// TwinCAT 3 PLC project Logger
// ProgramVersion: 3.1.4023.0
// libraries:
//   Tc2_Standard, * (Beckhoff Automation GmbH)
//   Tc2_System, * (Beckhoff Automation GmbH)
//   Tc2_Utilities, * (Beckhoff Automation GmbH)
//   Tc3_Module, * (Beckhoff Automation GmbH)
// project tree:
//   / PlcTask.TcTTO
//   POUs/ Logger.TcPOU, MAIN.TcPOU, Notifier.TcPOU, NotifierEvent.TcPOU
// real-time tasks:
//   TASK PlcTask: cycle T#10ms, priority 20, ADS port 350

CONFIGURATION Logger
    RESOURCE PLC ON TwinCAT3
        TASK PlcTask(INTERVAL := T#10ms, PRIORITY := 20);
        PROGRAM MAIN WITH PlcTask : MAIN;
    END_RESOURCE
END_CONFIGURATION

// ---- POUs/MAIN.TcPOU
PROGRAM MAIN
VAR
	
	diStep : DINT;
	bStart : BOOL;
	bStop : BOOL;
	fbRepeatTimer : TON;
	udiCounter : UDINT;
	
	fbLogger : Logger:= (sPathName:='C:\Users\fboid\Documents\ScopeTest\Log.txt');
	fbNotifier : Notifier := (sPathName:='C:\Users\fboid\Documents\ScopeTest\Log.csv');
	fbNotifierEvent : NotifierEvent;
	i : INT;
	bExecute : BOOL;
	uiCounter : UINT:= 0;
	bMotorError : BOOL;
	
END_VAR


//fbRepeatTimer(IN:= , PT:= T#5S, Q=> , ET=> );

fbNotifier(bExecute := bExecute);
fbNotifierEvent(
	CLK:= bMotorError,  
	fbNotifier:= fbNotifier, 
	sModuleName := 'PreHeat',
	sDeviceName := 'Load conveyor',
	sStatus := 'Error',
	sMessage := 'Motor overloaded');

END_PROGRAM

// ---- POUs/Logger.TcPOU
FUNCTION_BLOCK Logger
VAR_INPUT
	bExecute : BOOL;
	sPathName : STRING;
END_VAR
VAR_OUTPUT
END_VAR
VAR
	aBuffer : ARRAY[1..cMaxBufferRange] OF T_MaxString;
	aWorkBuffer : ARRAY[1..cMaxBufferRange] OF T_MaxString;
	aEmptyBuffer : ARRAY[1..cMaxBufferRange] OF T_MaxString; 
	
	fbFileWrite : FB_FileWrite;
	udiBufferCounter : UDINT;
	udiWorkCounter : UDINT;
	hFile : UINT;	
	
	fbFileOpen : FB_FileOpen;
	fbFilePuts : FB_FilePuts;
	fbFileClose : FB_FileClose;
	
	fbGetSystemTime : GETSYSTEMTIME;
	fbRepeatTimer : TON;
	diStep  : DINT;
	i : UDINT;
	bFilePutsIdle : BOOL;
	bExecuteFilePuts : BOOL;
	bInit : BOOL;
END_VAR
VAR CONSTANT
	cMaxBufferRange : UDINT := 1000;
END_VAR

fbFileOpen(
	sNetId:= , 
	sPathName:= sPathName,
	nMode:= FOPEN_MODEAPPEND OR FOPEN_MODETEXT, 
	ePath:= , 
	bExecute:=, 
	tTimeout:= , 
	bBusy=> , 
	bError=> , 
	nErrId=> , 
	hFile=> hFile);

fbFileWrite(
	sNetId:= , 
	hFile:= hFile, 
	pWriteBuff:= ADR(aWorkBuffer) , 
	cbWriteLen:= , 
	bExecute:= , 
	tTimeout:= , 
	bBusy=> , 
	bError=> , 
	nErrId=> , 
	cbWrite=> );

fbFileClose(
	sNetId:= , 
	hFile:= hFile, 
	bExecute:= , 
	tTimeout:= , 
	bBusy=> , 
	bError=> , 
	nErrId=> );
	
fbRepeatTimer(IN:= , PT:= T#2S, Q=> , ET=> );
//fbTime();

IF NOT bInit
THEN
	bInit := TRUE;
	FOR i := 1 TO cMaxBufferRange DO
		aEmptyBuffer[i] := '';
		aBuffer[i] := '';
		aWorkBuffer[i] := '';
	END_FOR
END_IF

IF 			bExecute
	AND  	diStep = 0
THEN
	diStep := 10;
END_IF	

CASE diStep OF
	
	10:
	
		fbFileOpen.bExecute := TRUE;
		fbRepeatTimer.IN := TRUE;
		diStep := 20;
		
	20:
	
		IF 		NOT fbFileOpen.bBusy
			AND NOT fbFIleOpen.bError
		THEN
			fbFileOpen.bExecute := FALSE;
			diStep := 30;
		END_IF
		
	30:
		
		IF udiBufferCounter > 0
		THEN
			udiWorkCounter := udiBufferCounter;
			udiBufferCounter := 0;
			
			aWorkBuffer := aBuffer;
			aBuffer := aEmptyBuffer;
			
			fbFileWrite.cbWriteLen := udiWorkCounter * (SIZEOF(T_MaxString));
			fbFileWrite.bExecute := TRUE;
			
			diStep := 40;
		ELSIF NOT bExecute
		THEN
			diStep := 50;
		END_IF
		
		
	40:
		
		IF NOT fbFileWrite.bBusy
		THEN
			
			fbFileWrite.bExecute := FALSE;
			IF fbRepeatTimer.Q
			THEN
				fbRepeatTImer.IN := FALSE;
				diStep := 50;
			ELSE
				diStep := 30;
			END_IF
			
		END_IF
		
	50:
	
		fbFileClose.bExecute := TRUE;
		diStep := 60;
		
	60: 
	
		IF 		NOT fbFileClose.bBusy
			AND NOT fbFileClose.bError
		THEN
			fbFileClose.bExecute := FALSE;
			IF bExecute 
			THEN
				
				diStep := 10;
			ELSE
				diStep := 0;
			END_IF
			
		END_IF
	
END_CASE

METHOD Write 
VAR_INPUT
	sMessage : T_MaxString;
END_VAR
VAR
	iLen : INT;
	iFillNumber : INT;
	i : INT;
	sTime : STRING;
	fileTime        : T_FILETIME;
END_VAR
IF udiBufferCounter < cMaxBufferRange
THEN

	udiBufferCounter := udiBufferCounter + 1;
	
	fbGetSystemTime(timeLoDW=>fileTime.dwLowDateTime, timeHiDW=>fileTime.dwHighDateTime );
	sTime :=SYSTEMTIME_TO_STRING( FILETIME_TO_SYSTEMTIME( fileTime ) );
	
	aBuffer[udiBufferCounter] := sTime;
	aBuffer[udiBufferCounter] := CONCAT(aBuffer[udiBufferCounter],': ');
	aBuffer[udiBufferCounter] := CONCAT(aBuffer[udiBufferCounter],sMessage);
	
	iLen := LEN(aBuffer[udiBufferCounter]);
	iFillNumber := 254-iLen;
	
	FOR i := 1 TO iFillNumber DO
		aBuffer[udiBufferCounter] := CONCAT(aBuffer[udiBufferCounter],' ');
	END_FOR
	
	aBuffer[udiBufferCounter][255] := F_ToAsc('$N');
	
END_IF
END_METHOD

END_FUNCTION_BLOCK

// ---- POUs/Notifier.TcPOU
FUNCTION_BLOCK Notifier
VAR_INPUT
	bExecute : BOOL;
	sPathName : STRING;
END_VAR
VAR_OUTPUT
END_VAR
VAR
	aBuffer : ARRAY[1..cMaxBufferRange] OF BYTE;
	aWorkBuffer : ARRAY[1..cMaxBufferRange] OF BYTE;
	aEmptyBuffer : ARRAY[1..cMaxBufferRange] OF BYTE; 
	
	fbFileWrite : FB_FileWrite;
	udiBufferCounter : UDINT;
	udiWorkCounter : UDINT;
	hFile : UINT;	
	
	fbFileOpen : FB_FileOpen;
	fbFilePuts : FB_FilePuts;
	fbFileClose : FB_FileClose;
	
	fbGetSystemTime : GETSYSTEMTIME;
	fbRepeatTimer : TON;
	diStep  : DINT;
	i : UDINT;
	bFilePutsIdle : BOOL;
	bExecuteFilePuts : BOOL;
	bInit : BOOL;
END_VAR
VAR CONSTANT
	cMaxBufferRange : UDINT := 1000 * 256;
END_VAR

fbFileOpen(
	sNetId:= , 
	sPathName:= sPathName,
	nMode:= FOPEN_MODEAPPEND OR FOPEN_MODETEXT, 
	ePath:= , 
	bExecute:=, 
	tTimeout:= , 
	bBusy=> , 
	bError=> , 
	nErrId=> , 
	hFile=> hFile);

fbFileWrite(
	sNetId:= , 
	hFile:= hFile, 
	pWriteBuff:= ADR(aWorkBuffer) , 
	cbWriteLen:= , 
	bExecute:= , 
	tTimeout:= , 
	bBusy=> , 
	bError=> , 
	nErrId=> , 
	cbWrite=> );

fbFileClose(
	sNetId:= , 
	hFile:= hFile, 
	bExecute:= , 
	tTimeout:= , 
	bBusy=> , 
	bError=> , 
	nErrId=> );
	
fbRepeatTimer(IN:= , PT:= T#2S, Q=> , ET=> );
//fbTime();

IF NOT bInit
THEN
	bInit := TRUE;
	(*
	FOR i := 1 TO cMaxBufferRange DO
		aEmptyBuffer[i] := '';
		aBuffer[i] := '';
		aWorkBuffer[i] := '';
	END_FOR
	*)
END_IF

IF 			bExecute
	AND  	diStep = 0
THEN
	diStep := 10;
END_IF	

CASE diStep OF
	
	10:
	
		fbFileOpen.bExecute := TRUE;
		fbRepeatTimer.IN := TRUE;
		diStep := 20;
		
	20:
	
		IF 		NOT fbFileOpen.bBusy
			AND NOT fbFIleOpen.bError
		THEN
			fbFileOpen.bExecute := FALSE;
			diStep := 30;
		END_IF
		
	30:
		
		IF udiBufferCounter > 0
		THEN
			udiWorkCounter := udiBufferCounter-1;
			udiBufferCounter := 0;
			
			aWorkBuffer := aBuffer;
			aBuffer := aEmptyBuffer;
			
			fbFileWrite.cbWriteLen := udiWorkCounter;
			fbFileWrite.bExecute := TRUE;
			
			diStep := 40;
		ELSIF NOT bExecute
		THEN
			diStep := 50;
		END_IF
		
		
	40:
		
		IF NOT fbFileWrite.bBusy
		THEN
			
			fbFileWrite.bExecute := FALSE;
			IF fbRepeatTimer.Q
			THEN
				fbRepeatTImer.IN := FALSE;
				diStep := 50;
			ELSE
				diStep := 30;
			END_IF
			
		END_IF
		
	50:
	
		fbFileClose.bExecute := TRUE;
		diStep := 60;
		
	60: 
	
		IF 		NOT fbFileClose.bBusy
			AND NOT fbFileClose.bError
		THEN
			fbFileClose.bExecute := FALSE;
			IF bExecute 
			THEN
				
				diStep := 10;
			ELSE
				diStep := 0;
			END_IF
			
		END_IF
	
END_CASE

METHOD Write 
VAR_INPUT
	
	sModuleName : T_MaxString;
	sDeviceName : T_MaxString;
	sStatus	: T_MaxString;
	sMessage : T_MaxString;
	
END_VAR
VAR
	iLen : INT;
	iFillNumber : INT;
	i : INT;
	sTime : STRING;
	fileTime : T_FILETIME;
	iTmpSize : INT;
	aLocalBuffer : ARRAY[0..MAX_STRING_LENGTH] OF BYTE;
	aEmptyLocalBuffer : ARRAY[0..MAX_STRING_LENGTH] OF BYTE;
END_VAR
IF udiBufferCounter < cMaxBufferRange
THEN
		
	fbGetSystemTime(timeLoDW=>fileTime.dwLowDateTime, timeHiDW=>fileTime.dwHighDateTime );
	sTime :=SYSTEMTIME_TO_STRING( FILETIME_TO_SYSTEMTIME( fileTime ) );

//Insert TimeStamp	
//----------------------------------------------------------------------------------------------------------------------------	
	iTmpSize := LEN(sTime);
	aLocalBuffer := MAXSTRING_TO_BYTEARR(sTime);
	
	FOR i:= 0 TO iTmpSize - 1 DO
		
		aBuffer[udiBufferCounter] := aLocalBuffer[i] ;	
		udiBufferCounter := udiBufferCounter + 1;
		
	END_FOR
//----------------------------------------------------------------------------------------------------------------------------
	
	aBuffer[udiBufferCounter] := F_ToAsc('$t');
	udiBufferCounter := udiBufferCounter + 1;
	
	aLocalBuffer := aEmptyLocalBuffer;

//Insert ModuleName	
//----------------------------------------------------------------------------------------------------------------------------	
	iTmpSize := LEN(sModuleName);
	aLocalBuffer := MAXSTRING_TO_BYTEARR(sModuleName);
	
	FOR i:= 0 TO iTmpSize - 1 DO
		
		aBuffer[udiBufferCounter] := aLocalBuffer[i] ;	
		udiBufferCounter := udiBufferCounter + 1;
		
	END_FOR
//----------------------------------------------------------------------------------------------------------------------------
	
	aBuffer[udiBufferCounter] := F_ToAsc('$t');
	udiBufferCounter := udiBufferCounter + 1;
	
	aLocalBuffer := aEmptyLocalBuffer;

//Insert DeviceName
//----------------------------------------------------------------------------------------------------------------------------
	iTmpSize := LEN(sDeviceName);
	aLocalBuffer := MAXSTRING_TO_BYTEARR(sDeviceName);
	
	FOR i:= 0 TO iTmpSize - 1 DO
		
		aBuffer[udiBufferCounter] := aLocalBuffer[i] ;	
		udiBufferCounter := udiBufferCounter + 1;
		
	END_FOR
//----------------------------------------------------------------------------------------------------------------------------	

	aBuffer[udiBufferCounter] := F_ToAsc('$t');
	udiBufferCounter := udiBufferCounter + 1;
	
	aLocalBuffer := aEmptyLocalBuffer;

//Insert Status
//----------------------------------------------------------------------------------------------------------------------------	
	iTmpSize := LEN(sStatus);
	aLocalBuffer := MAXSTRING_TO_BYTEARR(sStatus);
	
	FOR i:= 0 TO iTmpSize - 1 DO
		
		aBuffer[udiBufferCounter] := aLocalBuffer[i] ;	
		udiBufferCounter := udiBufferCounter + 1;
		
	END_FOR
//----------------------------------------------------------------------------------------------------------------------------
	
	aBuffer[udiBufferCounter] := F_ToAsc('$t');
	udiBufferCounter := udiBufferCounter + 1;
	
	aLocalBuffer := aEmptyLocalBuffer;

//Insert Message
//----------------------------------------------------------------------------------------------------------------------------	
	iTmpSize := LEN(sMessage);
	aLocalBuffer := MAXSTRING_TO_BYTEARR(sMessage);
	
	FOR i:= 0 TO iTmpSize - 1 DO
		
		aBuffer[udiBufferCounter] := aLocalBuffer[i] ;	
		udiBufferCounter := udiBufferCounter + 1;
		
	END_FOR	
//----------------------------------------------------------------------------------------------------------------------------
aBuffer[udiBufferCounter] := F_ToAsc('$N');
udiBufferCounter := udiBufferCounter + 1;	
	
END_IF
END_METHOD

END_FUNCTION_BLOCK

// ---- POUs/NotifierEvent.TcPOU
FUNCTION_BLOCK NotifierEvent EXTENDS R_TRIG
VAR_INPUT
	sModuleName : T_MaxString;
	sDeviceName : T_MaxString;
	sStatus: T_MaxString;
	sMessage : T_MaxString;
END_VAR
VAR_IN_OUT
	fbNotifier : Notifier;
END_VAR
VAR_OUTPUT
END_VAR
VAR
	
END_VAR

SUPER^();
IF 		Q
	AND __ISVALIDREF(fbNotifier)
THEN
	fbNotifier.Write(
		sDeviceName := sDeviceName,
		sMessage := sMessage,
		sModuleName := sModuleName,
		sStatus := sStatus);
END_IF

END_FUNCTION_BLOCK
